(* PLC project Untitled1, Eclipse Foundation CIF to Structured Text 0.0 *)
(* stored: creationDateTime 1970-01-01T00:00:00Z *)

TYPE TupleStruct : STRUCT
  field1 : DINT;
  field2 : DINT;
END_STRUCT;
END_TYPE

TYPE aut_location : (aut_l1, aut_l2);
END_TYPE

PROGRAM MAIN
  VAR
    inp : LREAL;
    c : LREAL;
    preset_c : TIME;
    aut_r : LREAL;
    aut_b : BOOL;
    aut_i : DINT;
    aut_tii : TupleStruct;
    aut_i2 : DINT;
    aut_i3 : DINT;
    aut : aut_location;
    firstRun : BOOL := TRUE;
  END_VAR
  VAR_TEMP
    curValue : LREAL;
    current_aut : aut_location;
    current_aut_b : BOOL;
    current_aut_i : DINT;
    current_aut_r : LREAL;
    current_aut_tii : TupleStruct;
    edge_aut_1 : DINT;
    eventEnabled : BOOL;
    ifResult : BOOL;
    isProgress : BOOL;
    litStruct : TupleStruct;
    timeOut : BOOL;
  END_VAR

            (* --- Initialize state or update continuous variables. -------------------- *)
IF firstRun THEN
    firstRun := FALSE;

    (* Initialize the state variables. *)
    c := 0.0;
    (* Reset timer of "c". *)
    preset_c := c;
    ton_c(IN := FALSE, PT := preset_c);
    ton_c(IN := TRUE, PT := preset_c);
    aut_r := 0.0;
    aut_b := FALSE;
    aut_i := 0;
    litStruct.field1 := 0;
    litStruct.field2 := 0;
    aut_tii := litStruct;
    aut_i2 := 1;
    aut_i3 := 1;
    aut := aut_l1;
ELSE
    (* Update remaining time of "c". *)
    ton_c(IN := TRUE, PT := preset_c, Q => timeOut, ET => curValue);
    c := SEL(timeOut, preset_c - curValue, 0.0);
END_IF;

(* --- Process uncontrollable events. -------------------------------------- *)
isProgress := TRUE;
(* Perform events until none can be done anymore. *)
WHILE isProgress DO
    isProgress := FALSE;

    (*************************************************************
     * Try to perform event "aut.f".
     *
     * - Automaton "aut" must always synchronize.
     *************************************************************)
    eventEnabled := TRUE;
    (*******************************
     * Check each synchronizing automaton for having an edge with a true guard.
     *******************************)
    (***********
     * Testing edges of automaton "aut" to synchronize for event "aut.f".
     * This automaton must have an edge with a true guard to allow the event.
     *
     * Edges being tested:
     * - Location "l1":
     *   - 36th edge in the location
     *   - 37th edge in the location
     ***********)
    IF aut = aut_l1 AND (aut_b OR aut_b) THEN
        edge_aut_1 := 1;
    ELSIF aut = aut_l1 AND aut_b THEN
        edge_aut_1 := 2;
    ELSE
        (* The automaton has no edge with a true guard. Skip to the next event. *)
        eventEnabled := FALSE;
    END_IF;
    (* All checks have been done. If variable "eventEnabled" still holds, event "aut.f" can occur. *)
    IF eventEnabled THEN
        isProgress := TRUE;
        (*******************************
         * Perform the assignments of each synchronizing automaton.
         *******************************)
        (* There are no assignments to perform for automata that must always synchronize. *)
        (* Automaton "aut" has no assignments to perform. *)
    END_IF;
END_WHILE;

(* --- Process controllable events. ---------------------------------------- *)
isProgress := TRUE;
(* Perform events until none can be done anymore. *)
WHILE isProgress DO
    isProgress := FALSE;

    (*************************************************************
     * Try to perform event "aut.e".
     *
     * - Automaton "aut" must always synchronize.
     *************************************************************)
    eventEnabled := TRUE;
    (*******************************
     * Check each synchronizing automaton for having an edge with a true guard.
     *******************************)
    (***********
     * Testing edges of automaton "aut" to synchronize for event "aut.e".
     * This automaton must have an edge with a true guard to allow the event.
     *
     * Edges being tested:
     * - Location "l1":
     *   - 1st edge in the location
     *   - 2nd edge in the location
     *   - 3rd edge in the location
     *   - 4th edge in the location
     *   - 5th edge in the location
     *   - 6th edge in the location
     *   - 7th edge in the location
     *   - 8th edge in the location
     *   - 9th edge in the location
     *   - 10th edge in the location
     *   - 11th edge in the location
     *   - 12th edge in the location
     *   - 13th edge in the location
     *   - 14th edge in the location
     *   - 15th edge in the location
     *   - 16th edge in the location
     *   - 17th edge in the location
     *   - 18th edge in the location
     *   - 19th edge in the location
     *   - 20th edge in the location
     *   - 21st edge in the location
     *   - 22nd edge in the location
     *   - 23rd edge in the location
     *   - 24th edge in the location
     *   - 25th edge in the location
     *   - 26th edge in the location
     *   - 27th edge in the location
     *   - 28th edge in the location
     *   - 29th edge in the location
     *   - 30th edge in the location
     *   - 31st edge in the location
     *   - 32nd edge in the location
     *   - 33rd edge in the location
     *   - 34th edge in the location
     *   - 35th edge in the location
     ***********)
    IF aut = aut_l1 THEN
        edge_aut_1 := 1;
    ELSIF aut = aut_l1 THEN
        edge_aut_1 := 2;
    ELSIF aut = aut_l1 THEN
        edge_aut_1 := 3;
    ELSIF aut = aut_l1 THEN
        edge_aut_1 := 4;
    ELSIF aut = aut_l1 THEN
        edge_aut_1 := 5;
    ELSIF aut = aut_l1 THEN
        edge_aut_1 := 6;
    ELSIF aut = aut_l1 THEN
        edge_aut_1 := 7;
    ELSIF aut = aut_l1 THEN
        edge_aut_1 := 8;
    ELSIF aut = aut_l1 THEN
        edge_aut_1 := 9;
    ELSIF aut = aut_l1 THEN
        edge_aut_1 := 10;
    ELSIF aut = aut_l1 THEN
        edge_aut_1 := 11;
    ELSIF aut = aut_l1 THEN
        edge_aut_1 := 12;
    ELSIF aut = aut_l1 THEN
        edge_aut_1 := 13;
    ELSIF aut = aut_l1 THEN
        edge_aut_1 := 14;
    ELSIF aut = aut_l1 THEN
        edge_aut_1 := 15;
    ELSIF aut = aut_l1 THEN
        edge_aut_1 := 16;
    ELSIF aut = aut_l1 THEN
        edge_aut_1 := 17;
    ELSIF aut = aut_l1 THEN
        edge_aut_1 := 18;
    ELSIF aut = aut_l1 THEN
        edge_aut_1 := 19;
    ELSIF aut = aut_l1 THEN
        edge_aut_1 := 20;
    ELSIF aut = aut_l1 THEN
        edge_aut_1 := 21;
    ELSIF aut = aut_l1 THEN
        edge_aut_1 := 22;
    ELSIF aut = aut_l1 THEN
        edge_aut_1 := 23;
    ELSIF aut = aut_l1 THEN
        edge_aut_1 := 24;
    ELSIF aut = aut_l1 THEN
        edge_aut_1 := 25;
    ELSIF aut = aut_l1 THEN
        edge_aut_1 := 26;
    ELSIF aut = aut_l1 THEN
        edge_aut_1 := 27;
    ELSIF aut = aut_l1 THEN
        edge_aut_1 := 28;
    ELSIF aut = aut_l1 THEN
        edge_aut_1 := 29;
    ELSIF aut = aut_l1 THEN
        edge_aut_1 := 30;
    ELSIF aut = aut_l1 THEN
        edge_aut_1 := 31;
    ELSIF aut = aut_l1 THEN
        edge_aut_1 := 32;
    ELSIF aut = aut_l1 THEN
        edge_aut_1 := 33;
    ELSIF aut = aut_l1 THEN
        edge_aut_1 := 34;
    ELSIF aut = aut_l1 THEN
        edge_aut_1 := 35;
    ELSE
        (* The automaton has no edge with a true guard. Skip to the next event. *)
        eventEnabled := FALSE;
    END_IF;
    (* All checks have been done. If variable "eventEnabled" still holds, event "aut.e" can occur. *)
    IF eventEnabled THEN
        isProgress := TRUE;
        (* Make temporary copies of assigned variables to preserve the old values while assigning new values. *)
        current_aut := aut;
        current_aut_b := aut_b;
        current_aut_i := aut_i;
        current_aut_r := aut_r;
        current_aut_tii := aut_tii;
        (*******************************
         * Perform the assignments of each synchronizing automaton.
         *******************************)
        (* Perform assignments of automaton "aut". *)
        IF edge_aut_1 = 1 THEN
            (* Perform assignments of the 1st edge in location "aut.l1". *)
            aut_r := inp;
        ELSIF edge_aut_1 = 2 THEN
            (* Perform assignments of the 2nd edge in location "aut.l1". *)
            aut_r := inp + -1.0;
            aut := aut_l2;
        ELSIF edge_aut_1 = 3 THEN
            (* Perform assignments of the 3rd edge in location "aut.l1". *)
            aut_r := DINT_TO_LREAL(current_aut_i);
        ELSIF edge_aut_1 = 4 THEN
            (* Perform assignments of the 4th edge in location "aut.l1". *)
            aut_b := NOT current_aut_b;
        ELSIF edge_aut_1 = 5 THEN
            (* Perform assignments of the 5th edge in location "aut.l1". *)
            aut_b := current_aut_b OR NOT current_aut_b;
        ELSIF edge_aut_1 = 6 THEN
            (* Perform assignments of the 6th edge in location "aut.l1". *)
            aut_r := DINT_TO_LREAL(current_aut_i) / DINT_TO_LREAL(current_aut_i);
        ELSIF edge_aut_1 = 7 THEN
            (* Perform assignments of the 7th edge in location "aut.l1". *)
            IF current_aut_b THEN
                ifResult := current_aut_b;
            ELSE
                ifResult := current_aut_b;
            END_IF;
            aut_b := ifResult;
        ELSIF edge_aut_1 = 8 THEN
            (* Perform assignments of the 8th edge in location "aut.l1". *)
            aut_i := current_aut_tii.field1;
        ELSIF edge_aut_1 = 9 THEN
            (* Perform assignments of the 9th edge in location "aut.l1". *)
            aut_r := ABS(current_aut_r);
        ELSIF edge_aut_1 = 10 THEN
            (* Perform assignments of the 10th edge in location "aut.l1". *)
            aut_r := current_aut_r ** (1.0 / 3.0);
        ELSIF edge_aut_1 = 11 THEN
            (* Perform assignments of the 11th edge in location "aut.l1". *)
            aut_r := EXP(current_aut_r);
        ELSIF edge_aut_1 = 12 THEN
            (* Perform assignments of the 12th edge in location "aut.l1". *)
            aut_r := LN(current_aut_r);
        ELSIF edge_aut_1 = 13 THEN
            (* Perform assignments of the 13th edge in location "aut.l1". *)
            aut_r := LOG(current_aut_r);
        ELSIF edge_aut_1 = 14 THEN
            (* Perform assignments of the 14th edge in location "aut.l1". *)
            aut_i := MIN(current_aut_i, current_aut_i);
        ELSIF edge_aut_1 = 15 THEN
            (* Perform assignments of the 15th edge in location "aut.l1". *)
            aut_r := MIN(DINT_TO_LREAL(current_aut_i), current_aut_r);
        ELSIF edge_aut_1 = 16 THEN
            (* Perform assignments of the 16th edge in location "aut.l1". *)
            aut_r := MIN(current_aut_r, DINT_TO_LREAL(current_aut_i));
        ELSIF edge_aut_1 = 17 THEN
            (* Perform assignments of the 17th edge in location "aut.l1". *)
            aut_r := MIN(current_aut_r, current_aut_r);
        ELSIF edge_aut_1 = 18 THEN
            (* Perform assignments of the 18th edge in location "aut.l1". *)
            aut_i := MAX(current_aut_i, current_aut_i);
        ELSIF edge_aut_1 = 19 THEN
            (* Perform assignments of the 19th edge in location "aut.l1". *)
            aut_r := MAX(DINT_TO_LREAL(current_aut_i), current_aut_r);
        ELSIF edge_aut_1 = 20 THEN
            (* Perform assignments of the 20th edge in location "aut.l1". *)
            aut_r := MAX(current_aut_r, DINT_TO_LREAL(current_aut_i));
        ELSIF edge_aut_1 = 21 THEN
            (* Perform assignments of the 21st edge in location "aut.l1". *)
            aut_r := MAX(current_aut_r, current_aut_r);
        ELSIF edge_aut_1 = 22 THEN
            (* Perform assignments of the 22nd edge in location "aut.l1". *)
            aut_i := LREAL_TO_DINT(DINT_TO_LREAL(aut_i2) ** aut_i3);
        ELSIF edge_aut_1 = 23 THEN
            (* Perform assignments of the 23rd edge in location "aut.l1". *)
            aut_r := DINT_TO_LREAL(current_aut_i) ** current_aut_i;
        ELSIF edge_aut_1 = 24 THEN
            (* Perform assignments of the 24th edge in location "aut.l1". *)
            aut_r := DINT_TO_LREAL(current_aut_i) ** current_aut_r;
        ELSIF edge_aut_1 = 25 THEN
            (* Perform assignments of the 25th edge in location "aut.l1". *)
            aut_r := current_aut_r ** current_aut_i;
        ELSIF edge_aut_1 = 26 THEN
            (* Perform assignments of the 26th edge in location "aut.l1". *)
            aut_r := current_aut_r ** current_aut_r;
        ELSIF edge_aut_1 = 27 THEN
            (* Perform assignments of the 27th edge in location "aut.l1". *)
            aut_r := SQRT(current_aut_r);
        ELSIF edge_aut_1 = 28 THEN
            (* Perform assignments of the 28th edge in location "aut.l1". *)
            aut_r := ASIN(current_aut_r);
        ELSIF edge_aut_1 = 29 THEN
            (* Perform assignments of the 29th edge in location "aut.l1". *)
            aut_r := ACOS(current_aut_r);
        ELSIF edge_aut_1 = 30 THEN
            (* Perform assignments of the 30th edge in location "aut.l1". *)
            aut_r := ATAN(current_aut_r);
        ELSIF edge_aut_1 = 31 THEN
            (* Perform assignments of the 31st edge in location "aut.l1". *)
            aut_r := SIN(current_aut_r);
        ELSIF edge_aut_1 = 32 THEN
            (* Perform assignments of the 32nd edge in location "aut.l1". *)
            aut_r := COS(current_aut_r);
        ELSIF edge_aut_1 = 33 THEN
            (* Perform assignments of the 33rd edge in location "aut.l1". *)
            aut_r := TAN(current_aut_r);
        ELSIF edge_aut_1 = 34 THEN
            (* Perform assignments of the 34th edge in location "aut.l1". *)
            litStruct.field1 := current_aut_i;
            litStruct.field2 := current_aut_i + 1;
            aut_tii := litStruct;
        ELSIF edge_aut_1 = 35 THEN
            (* Perform assignments of the 35th edge in location "aut.l1". *)
            aut_r := current_aut_r * 2.0;
            aut_i := current_aut_i + 1;
        END_IF;
    END_IF;
END_WHILE;
          
END_PROGRAM

CONFIGURATION Untitled1
  RESOURCE Untitled1 ON PLC
    VAR_GLOBAL  (* TIMERS *)
      ton_c : TON;
    END_VAR
    TASK PlcTask(INTERVAL := T#10ms, PRIORITY := 20);
    PROGRAM MAIN WITH PlcTask : MAIN;
  END_RESOURCE
END_CONFIGURATION
